TYPE "HMI_Preset"
VERSION : 0.1
// Block: HMI_Preset
   STRUCT
      Button : Bool;
      Value : LReal;
      Feedback : LReal;
   END_STRUCT;

END_TYPE
